(*********************************** G.D S.p.A. - Technical Department ***********************************
============= PROGRAM INFO ============
FOLDER:             TBD
MACHINES INVOLVED:  TBD 

============= DESCRIPTION =============
csp machine declaration

============= REVISIONS ===============
Date		Version	 	Author      	Description             
----------	-------		------------  	--------------------------------------------
2019/04/05 	0000.00	 	M.Grasso		Creation of the PRG

**********************************************************************************************************)
(*$R process_ref := prc; $*)
PROGRAM csp_case_discharge_speedBelt
VAR
		
	prc:											process;
	prc_path:										STRING;
	
END_VAR

_read_var_input();

_object_manager();

IF NOT objects_running()
THEN
	RETURN;	
END_IF

_read_process_image();

_mode_manager();

_set_runtime_properties();

(********************************* BODY *********************************)
(************************************************************************)

_handle_messages();

_write_output();

ACTION _handle_messages:
;
END_ACTION

ACTION _handle_process_test:
;
END_ACTION

ACTION _mode_manager:
IF process_mode_req_is_pending(prc)
THEN
    process_apply_mode_req_first_step(prc);
    CASE process_get_mode(prc) OF
        MODE_TO_ABSENT:
			;
        MODE_TO_INACTIVE:
			;
        MODE_TO_TEST:
			;
        MODE_TO_OPERATIONAL:
			;
    END_CASE
    process_apply_mode_req_second_step(prc);
END_IF
END_ACTION

ACTION _object_manager:
IF objects_initialization()
THEN
	sub_process_init(
		object_name					:= 'csp_case_discharge_speedBelt.prc', 
		process						:= csp_case_discharge.prc, 
		CONVERSION_this				:= prc);
		
	prc_path 						:= process_get_path(prc);
END_IF

IF objects_running()
THEN
	process_cycle(prc);
END_IF
END_ACTION

ACTION _read_process_image:
;
END_ACTION

ACTION _read_var_input:
;
END_ACTION

ACTION _set_runtime_properties:
;
END_ACTION

ACTION _write_output:
;
END_ACTION

END_PROGRAM

(* stored: Version 1.1.0.1, ProductVersion 3.1.4022.12
   POU csp_case_discharge_speedBelt: Id {6ba4e706-4034-477f-9a02-ac85f7223e21}, SpecialFunc None
   Action _handle_messages: Id {3b13bb4c-2fc3-42a3-92ec-0c5a49eaa839}
   Action _handle_process_test: Id {410e716e-3f35-44c5-9035-e24495d027ec}
   Action _mode_manager: Id {6ba69840-79a5-4b57-94fc-5f8b0213f3e8}
   Action _object_manager: Id {acd16ade-3187-4aa9-a008-54b70a909112}
   Action _read_process_image: Id {9b2bcf7d-cbf6-4220-ac96-f6444cb50dec}
   Action _read_var_input: Id {40fe982b-a75e-4072-a8a5-fbdac8b80b49}
   Action _set_runtime_properties: Id {73d68e32-0fb2-4c08-b945-05829eaee06e}
   Action _write_output: Id {2a351f82-b318-4b9b-9e3a-f73f60682f1f} *)
